// TIA Portal V20 export
DATA_BLOCK "AirConditioner_DB"   // DB549
// stored: AutoNumber false, InstanceOfName AirConditioner, InstanceOfType FB
"AirConditioner"
   // VAR
   //    Var : "TypeVar";
   //    T : Array[1..4] of IEC_TIMER;
   //    air1Active : Bool;
   //    air1InputNo : Bool;
   //    air2Active : Bool;
   //    air2InputNo : Bool;
   //    airXrayActive : Bool;
   //    airXrayInputNo : Bool;
   //    airDehActive : Bool;
   //    airDehInputNo : Bool;
   // END_VAR
BEGIN
END_DATA_BLOCK
